// Mitsubishi GX Works2 project: may ver1   PLC: FX3G

PROGRAM MAIN
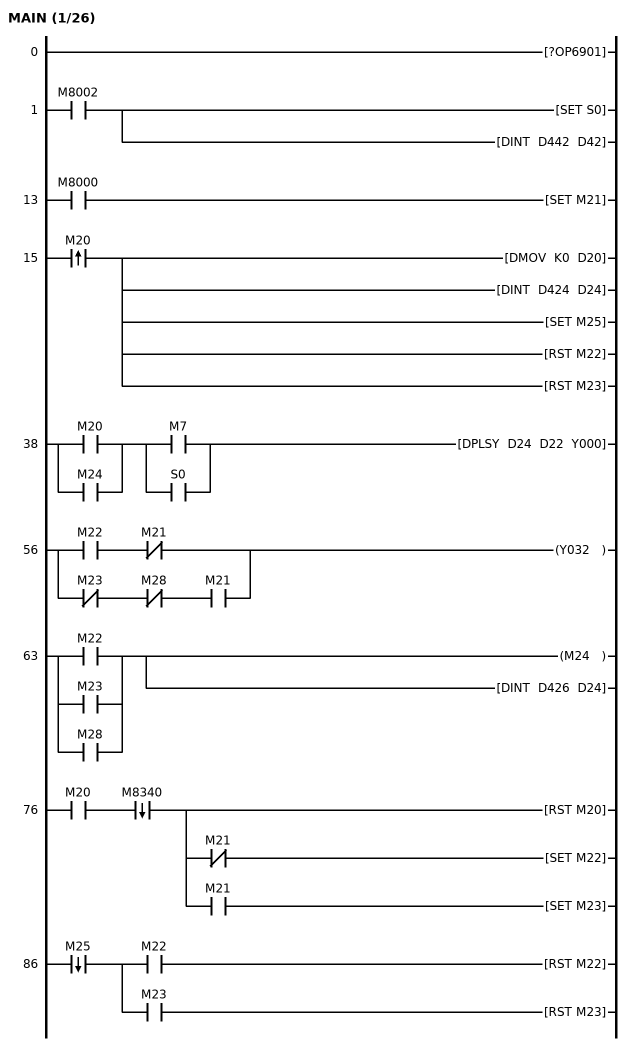
0     ?OP6901
1     LD      M8002
      SET     S0
      DINT    D442 D42
13    LD      M8000
      SET     M21
15    LDP     M20
      DMOV    K0 D20
      DINT    D424 D24
      SET     M25
      RST     M22
      RST     M23
38    LD      M20
      OR      M24
      LD      M7
      OR      S0
      ANB
      DPLSY   D24 D22 Y000
56    LD      M22
      ANI     M21
      LDI     M23
      ANI     M28
      AND     M21
      ORB
      OUT     Y032
63    LD      M22
      OR      M23
      OR      M28
      OUT     M24
      DINT    D426 D24
76    LD      M20
      ANDF    M8340
      RST     M20
      MPS
      ANI     M21
      SET     M22
      MPP
      AND     M21
      SET     M23
86    LDF     M25
      MPS
      AND     M22
      RST     M22
      MPP
      AND     M23
      RST     M23
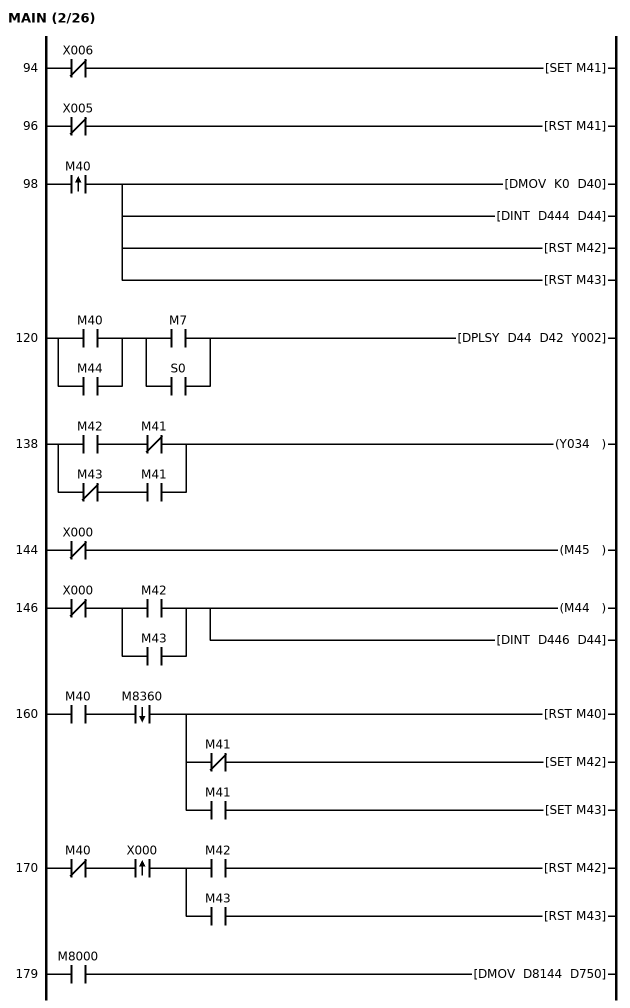
94    LDI     X006
      SET     M41
96    LDI     X005
      RST     M41
98    LDP     M40
      DMOV    K0 D40
      DINT    D444 D44
      RST     M42
      RST     M43
120   LD      M40
      OR      M44
      LD      M7
      OR      S0
      ANB
      DPLSY   D44 D42 Y002
138   LD      M42
      ANI     M41
      LDI     M43
      AND     M41
      ORB
      OUT     Y034
144   LDI     X000
      OUT     M45
146   LDI     X000
      LD      M42
      OR      M43
      ANB
      OUT     M44
      DINT    D446 D44
160   LD      M40
      ANDF    M8360
      RST     M40
      MPS
      ANI     M41
      SET     M42
      MPP
      AND     M41
      SET     M43
170   LDI     M40
      ANDP    X000
      MPS
      AND     M42
      RST     M42
      MPP
      AND     M43
      RST     M43
179   LD      M8000
      DMOV    D8144 D750
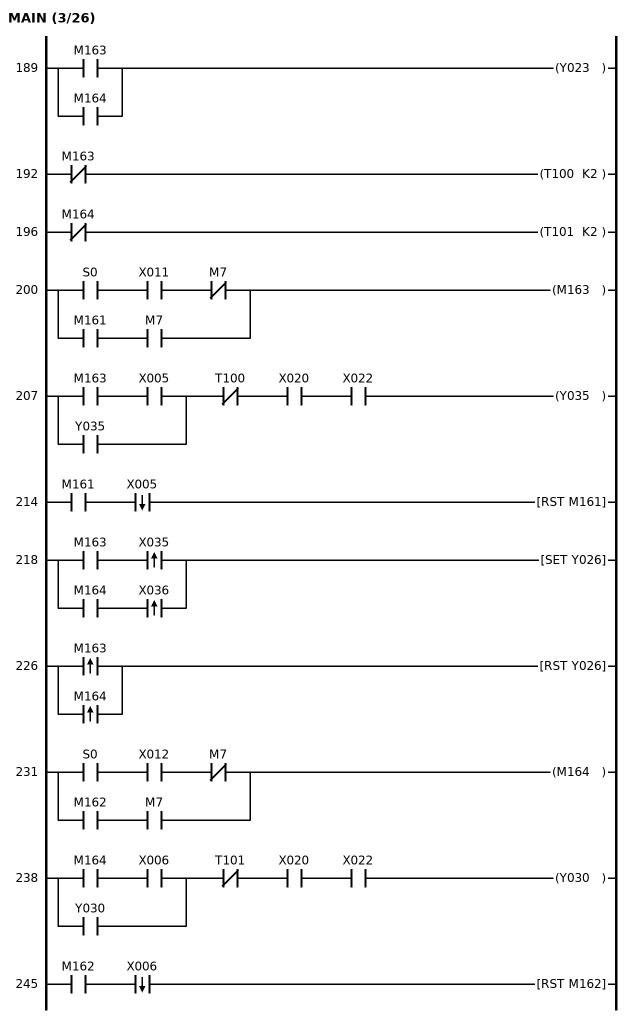
189   LD      M163
      OR      M164
      OUT     Y023
192   LDI     M163
      OUT     T100 K2
196   LDI     M164
      OUT     T101 K2
200   LD      S0
      AND     X011
      ANI     M7
      LD      M161
      AND     M7
      ORB
      OUT     M163
207   LD      M163
      AND     X005
      OR      Y035
      ANI     T100
      AND     X020
      AND     X022
      OUT     Y035
214   LD      M161
      ANDF    X005
      RST     M161
218   LD      M163
      ANDP    X035
      LD      M164
      ANDP    X036
      ORB
      SET     Y026
226   LDP     M163
      ORP     M164
      RST     Y026
231   LD      S0
      AND     X012
      ANI     M7
      LD      M162
      AND     M7
      ORB
      OUT     M164
238   LD      M164
      AND     X006
      OR      Y030
      ANI     T101
      AND     X020
      AND     X022
      OUT     Y030
245   LD      M162
      ANDF    X006
      RST     M162
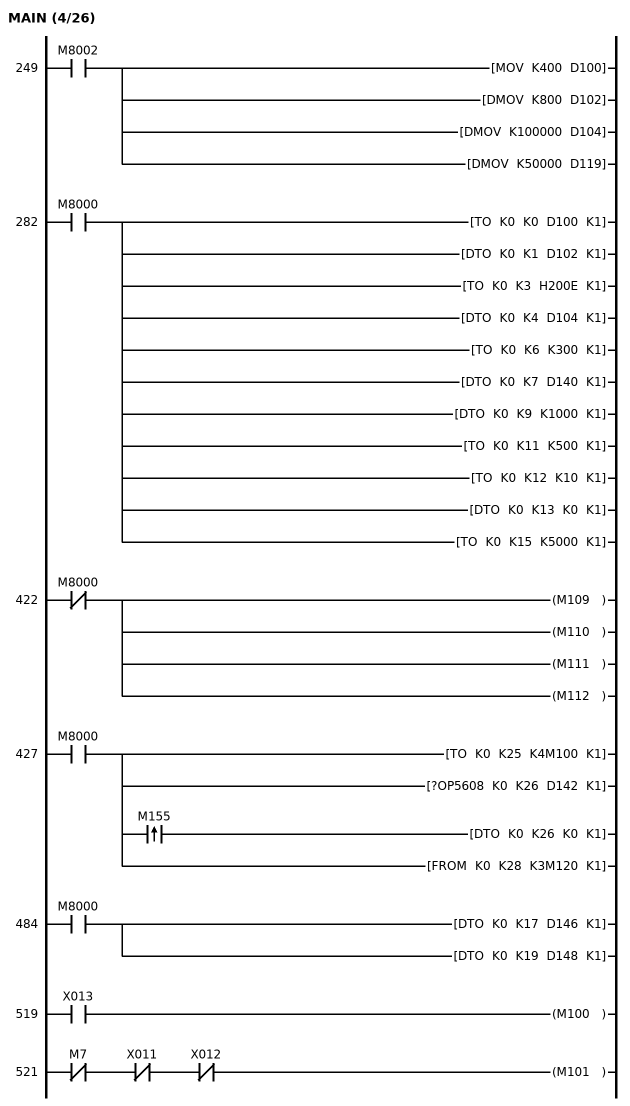
249   LD      M8002
      MOV     K400 D100
      DMOV    K800 D102
      DMOV    K100000 D104
      DMOV    K50000 D119
282   LD      M8000
      TO      K0 K0 D100 K1
      DTO     K0 K1 D102 K1
      TO      K0 K3 H200E K1
      DTO     K0 K4 D104 K1
      TO      K0 K6 K300 K1
      DTO     K0 K7 D140 K1
      DTO     K0 K9 K1000 K1
      TO      K0 K11 K500 K1
      TO      K0 K12 K10 K1
      DTO     K0 K13 K0 K1
      TO      K0 K15 K5000 K1
422   LDI     M8000
      OUT     M109
      OUT     M110
      OUT     M111
      OUT     M112
427   LD      M8000
      TO      K0 K25 K4M100 K1
      ?OP5608 K0 K26 D142 K1
      MPS
      ANDP    M155
      DTO     K0 K26 K0 K1
      MPP
      FROM    K0 K28 K3M120 K1
484   LD      M8000
      DTO     K0 K17 D146 K1
      DTO     K0 K19 D148 K1
519   LD      X013
      OUT     M100
521   LDI     M7
      ANI     X011
      ANI     X012
      OUT     M101
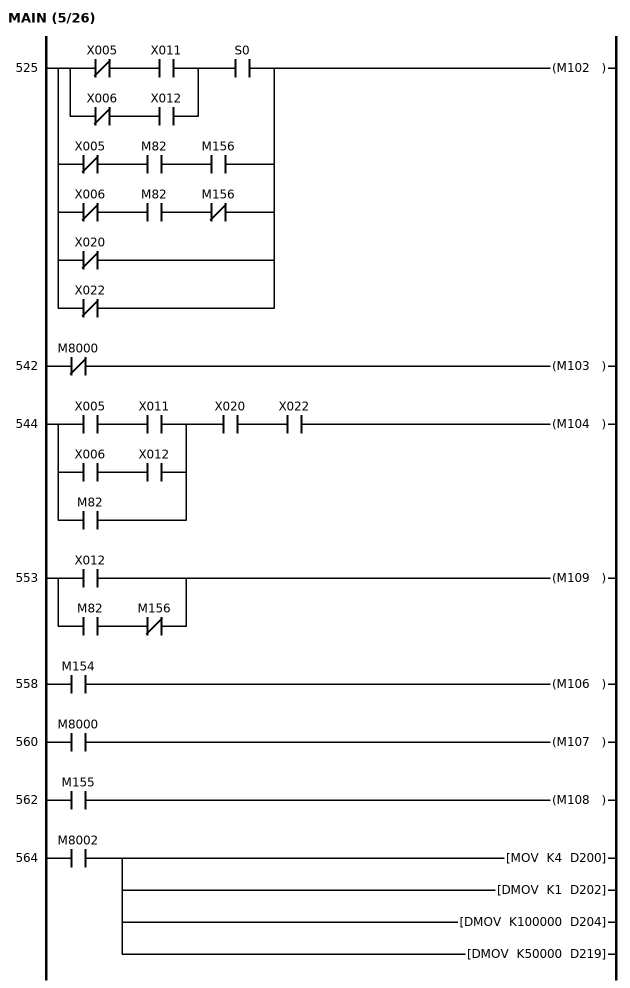
525   LDI     X005
      AND     X011
      LDI     X006
      AND     X012
      ORB
      AND     S0
      LDI     X005
      AND     M82
      AND     M156
      ORB
      LDI     X006
      AND     M82
      ANI     M156
      ORB
      ORI     X020
      ORI     X022
      OUT     M102
542   LDI     M8000
      OUT     M103
544   LD      X005
      AND     X011
      LD      X006
      AND     X012
      ORB
      OR      M82
      AND     X020
      AND     X022
      OUT     M104
553   LD      X012
      LD      M82
      ANI     M156
      ORB
      OUT     M109
558   LD      M154
      OUT     M106
560   LD      M8000
      OUT     M107
562   LD      M155
      OUT     M108
564   LD      M8002
      MOV     K4 D200
      DMOV    K1 D202
      DMOV    K100000 D204
      DMOV    K50000 D219
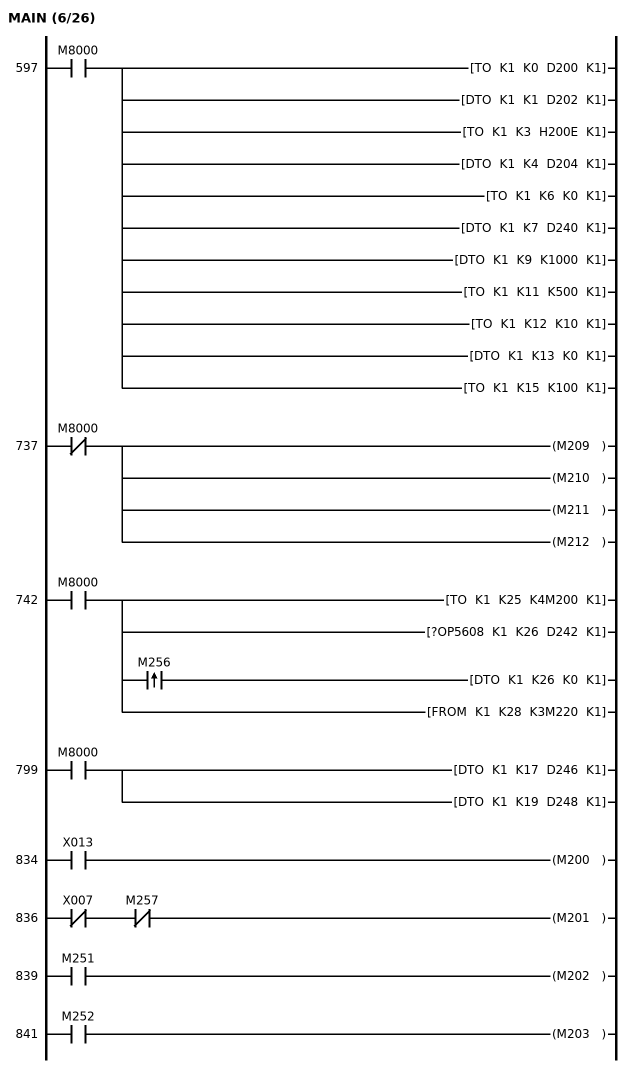
597   LD      M8000
      TO      K1 K0 D200 K1
      DTO     K1 K1 D202 K1
      TO      K1 K3 H200E K1
      DTO     K1 K4 D204 K1
      TO      K1 K6 K0 K1
      DTO     K1 K7 D240 K1
      DTO     K1 K9 K1000 K1
      TO      K1 K11 K500 K1
      TO      K1 K12 K10 K1
      DTO     K1 K13 K0 K1
      TO      K1 K15 K100 K1
737   LDI     M8000
      OUT     M209
      OUT     M210
      OUT     M211
      OUT     M212
742   LD      M8000
      TO      K1 K25 K4M200 K1
      ?OP5608 K1 K26 D242 K1
      MPS
      ANDP    M256
      DTO     K1 K26 K0 K1
      MPP
      FROM    K1 K28 K3M220 K1
799   LD      M8000
      DTO     K1 K17 D246 K1
      DTO     K1 K19 D248 K1
834   LD      X013
      OUT     M200
836   LDI     X007
      ANI     M257
      OUT     M201
839   LD      M251
      OUT     M202
841   LD      M252
      OUT     M203
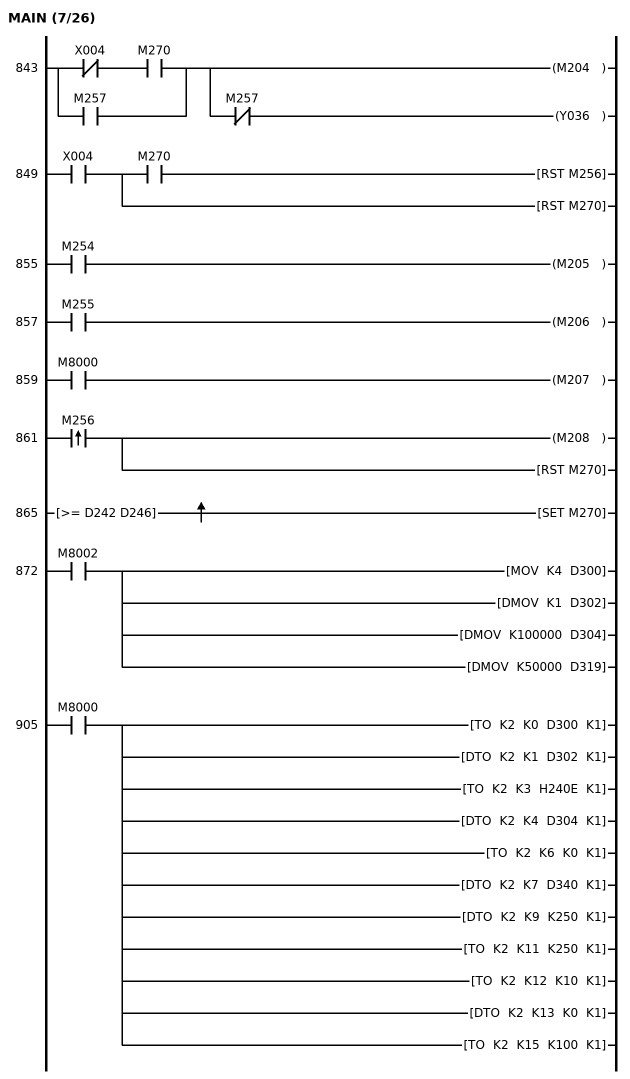
843   LDI     X004
      AND     M270
      OR      M257
      OUT     M204
      ANI     M257
      OUT     Y036
849   LD      X004
      MPS
      AND     M270
      RST     M256
      MPP
      RST     M270
855   LD      M254
      OUT     M205
857   LD      M255
      OUT     M206
859   LD      M8000
      OUT     M207
861   LDP     M256
      OUT     M208
      RST     M270
865   LD>=    D242 D246
      MEP
      SET     M270
872   LD      M8002
      MOV     K4 D300
      DMOV    K1 D302
      DMOV    K100000 D304
      DMOV    K50000 D319
905   LD      M8000
      TO      K2 K0 D300 K1
      DTO     K2 K1 D302 K1
      TO      K2 K3 H240E K1
      DTO     K2 K4 D304 K1
      TO      K2 K6 K0 K1
      DTO     K2 K7 D340 K1
      DTO     K2 K9 K250 K1
      TO      K2 K11 K250 K1
      TO      K2 K12 K10 K1
      DTO     K2 K13 K0 K1
      TO      K2 K15 K100 K1
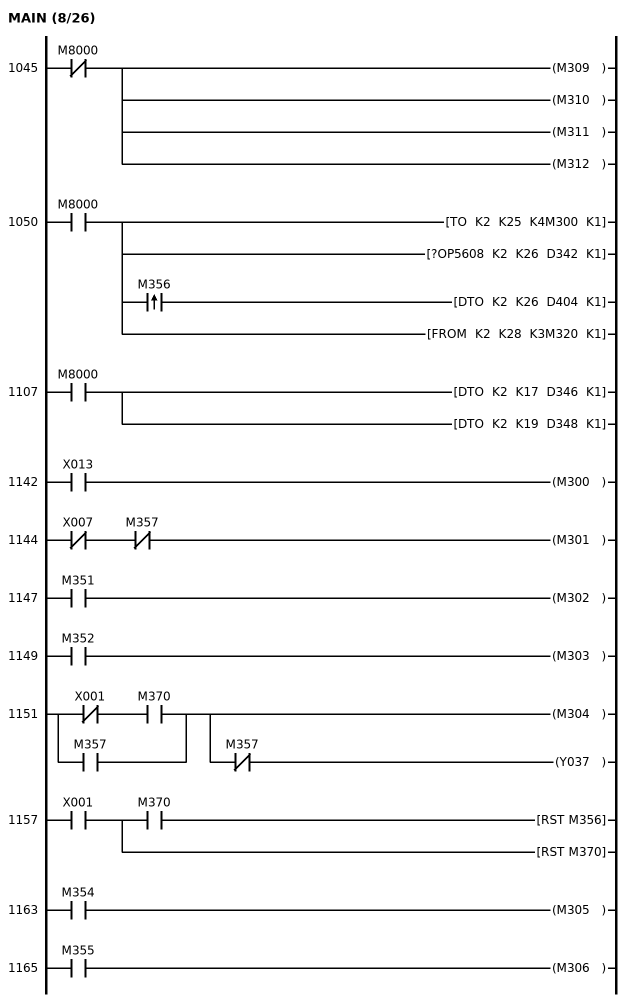
1045  LDI     M8000
      OUT     M309
      OUT     M310
      OUT     M311
      OUT     M312
1050  LD      M8000
      TO      K2 K25 K4M300 K1
      ?OP5608 K2 K26 D342 K1
      MPS
      ANDP    M356
      DTO     K2 K26 D404 K1
      MPP
      FROM    K2 K28 K3M320 K1
1107  LD      M8000
      DTO     K2 K17 D346 K1
      DTO     K2 K19 D348 K1
1142  LD      X013
      OUT     M300
1144  LDI     X007
      ANI     M357
      OUT     M301
1147  LD      M351
      OUT     M302
1149  LD      M352
      OUT     M303
1151  LDI     X001
      AND     M370
      OR      M357
      OUT     M304
      ANI     M357
      OUT     Y037
1157  LD      X001
      MPS
      AND     M370
      RST     M356
      MPP
      RST     M370
1163  LD      M354
      OUT     M305
1165  LD      M355
      OUT     M306
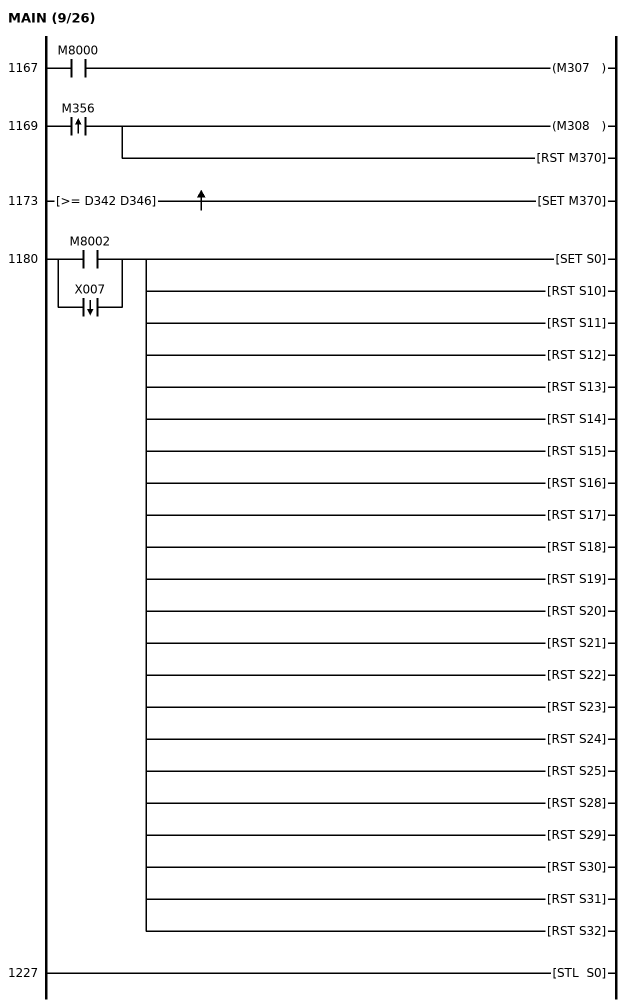
1167  LD      M8000
      OUT     M307
1169  LDP     M356
      OUT     M308
      RST     M370
1173  LD>=    D342 D346
      MEP
      SET     M370
1180  LD      M8002
      ORF     X007
      SET     S0
      RST     S10
      RST     S11
      RST     S12
      RST     S13
      RST     S14
      RST     S15
      RST     S16
      RST     S17
      RST     S18
      RST     S19
      RST     S20
      RST     S21
      RST     S22
      RST     S23
      RST     S24
      RST     S25
      RST     S28
      RST     S29
      RST     S30
      RST     S31
      RST     S32
1227  STL     S0
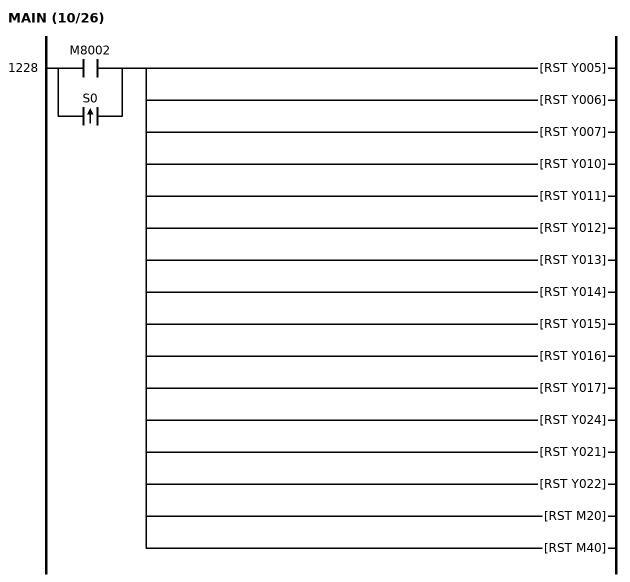
1228  LD      M8002
      ORP     S0
      RST     Y005
      RST     Y006
      RST     Y007
      RST     Y010
      RST     Y011
      RST     Y012
      RST     Y013
      RST     Y014
      RST     Y015
      RST     Y016
      RST     Y017
      RST     Y024
      RST     Y021
      RST     Y022
      RST     M20
      RST     M40
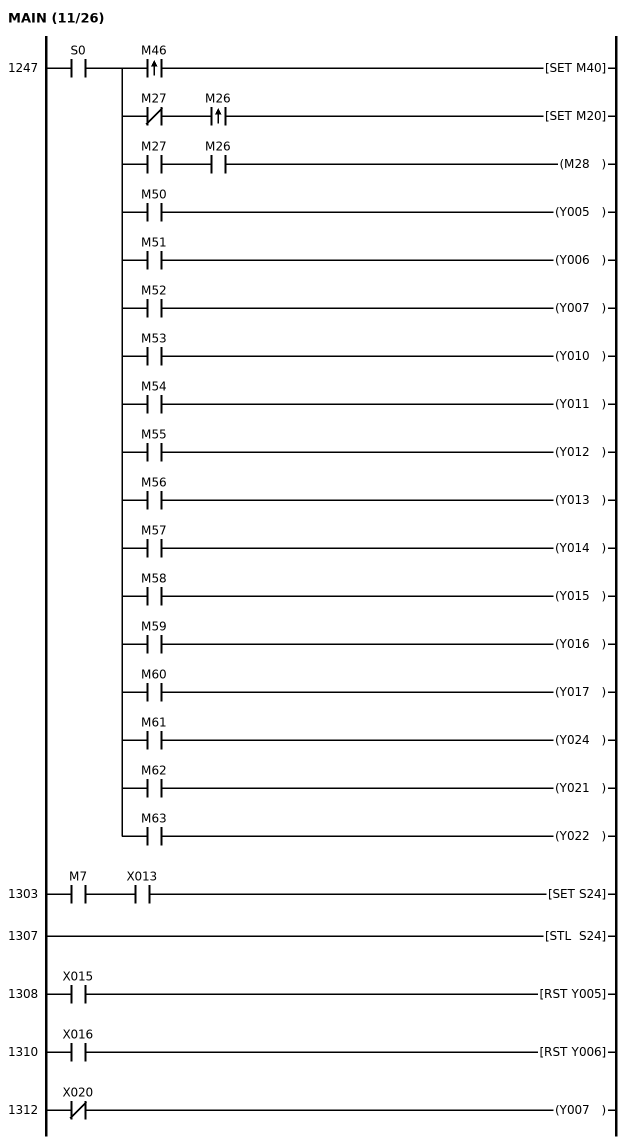
1247  LD      S0
      MPS
      ANDP    M46
      SET     M40
      MRD
      ANI     M27
      ANDP    M26
      SET     M20
      MRD
      AND     M27
      AND     M26
      OUT     M28
      MRD
      AND     M50
      OUT     Y005
      MRD
      AND     M51
      OUT     Y006
      MRD
      AND     M52
      OUT     Y007
      MRD
      AND     M53
      OUT     Y010
      MRD
      AND     M54
      OUT     Y011
      MRD
      AND     M55
      OUT     Y012
      MRD
      AND     M56
      OUT     Y013
      MRD
      AND     M57
      OUT     Y014
      MRD
      AND     M58
      OUT     Y015
      MRD
      AND     M59
      OUT     Y016
      MRD
      AND     M60
      OUT     Y017
      MRD
      AND     M61
      OUT     Y024
      MRD
      AND     M62
      OUT     Y021
      MPP
      AND     M63
      OUT     Y022
1303  LD      M7
      AND     X013
      SET     S24
1307  STL     S24
1308  LD      X015
      RST     Y005
1310  LD      X016
      RST     Y006
1312  LDI     X020
      OUT     Y007
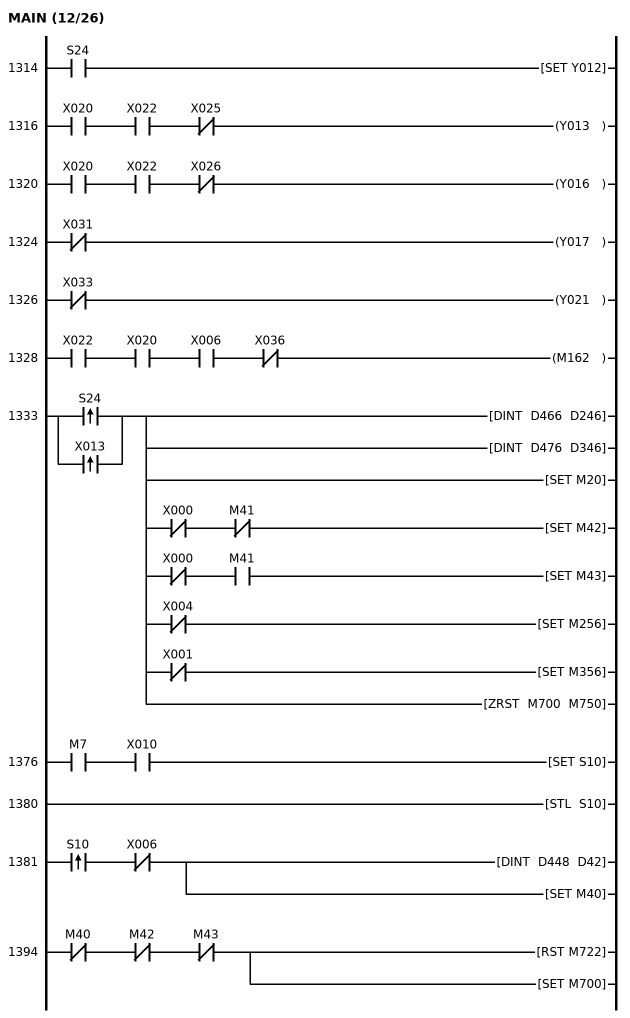
1314  LD      S24
      SET     Y012
1316  LD      X020
      AND     X022
      ANI     X025
      OUT     Y013
1320  LD      X020
      AND     X022
      ANI     X026
      OUT     Y016
1324  LDI     X031
      OUT     Y017
1326  LDI     X033
      OUT     Y021
1328  LD      X022
      AND     X020
      AND     X006
      ANI     X036
      OUT     M162
1333  LDP     S24
      ORP     X013
      DINT    D466 D246
      DINT    D476 D346
      SET     M20
      MPS
      ANI     X000
      ANI     M41
      SET     M42
      MRD
      ANI     X000
      AND     M41
      SET     M43
      MRD
      ANI     X004
      SET     M256
      MRD
      ANI     X001
      SET     M356
      MPP
      ZRST    M700 M750
1376  LD      M7
      AND     X010
      SET     S10
1380  STL     S10
1381  LDP     S10
      ANI     X006
      DINT    D448 D42
      SET     M40
1394  LDI     M40
      ANI     M42
      ANI     M43
      RST     M722
      SET     M700
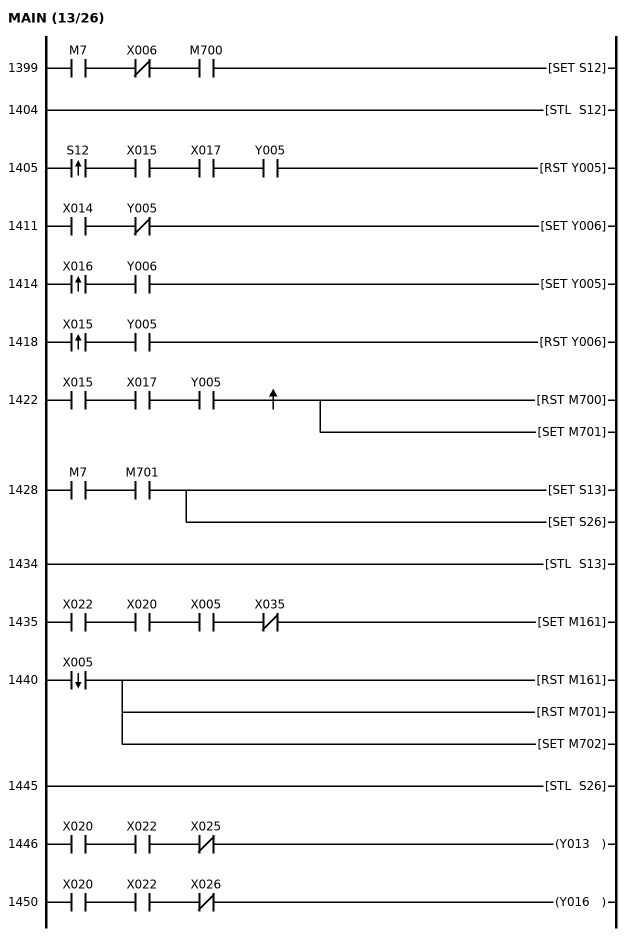
1399  LD      M7
      ANI     X006
      AND     M700
      SET     S12
1404  STL     S12
1405  LDP     S12
      AND     X015
      AND     X017
      AND     Y005
      RST     Y005
1411  LD      X014
      ANI     Y005
      SET     Y006
1414  LDP     X016
      AND     Y006
      SET     Y005
1418  LDP     X015
      AND     Y005
      RST     Y006
1422  LD      X015
      AND     X017
      AND     Y005
      MEP
      RST     M700
      SET     M701
1428  LD      M7
      AND     M701
      SET     S13
      SET     S26
1434  STL     S13
1435  LD      X022
      AND     X020
      AND     X005
      ANI     X035
      SET     M161
1440  LDF     X005
      RST     M161
      RST     M701
      SET     M702
1445  STL     S26
1446  LD      X020
      AND     X022
      ANI     X025
      OUT     Y013
1450  LD      X020
      AND     X022
      ANI     X026
      OUT     Y016
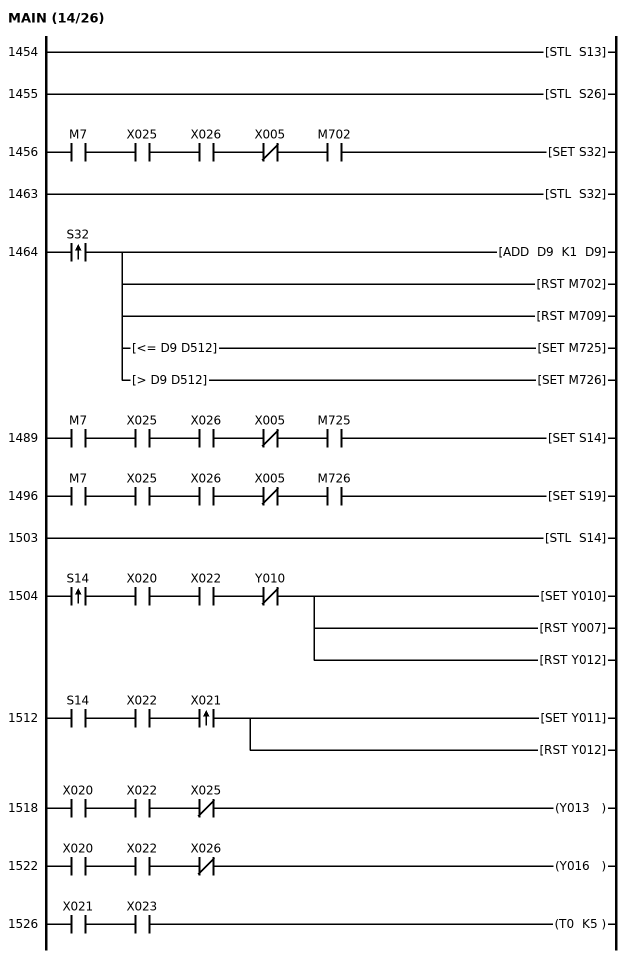
1454  STL     S13
1455  STL     S26
1456  LD      M7
      AND     X025
      AND     X026
      ANI     X005
      AND     M702
      SET     S32
1463  STL     S32
1464  LDP     S32
      ADD     D9 K1 D9
      RST     M702
      RST     M709
      MPS
      AND<=   D9 D512
      SET     M725
      MPP
      AND>    D9 D512
      SET     M726
1489  LD      M7
      AND     X025
      AND     X026
      ANI     X005
      AND     M725
      SET     S14
1496  LD      M7
      AND     X025
      AND     X026
      ANI     X005
      AND     M726
      SET     S19
1503  STL     S14
1504  LDP     S14
      AND     X020
      AND     X022
      ANI     Y010
      SET     Y010
      RST     Y007
      RST     Y012
1512  LD      S14
      AND     X022
      ANDP    X021
      SET     Y011
      RST     Y012
1518  LD      X020
      AND     X022
      ANI     X025
      OUT     Y013
1522  LD      X020
      AND     X022
      ANI     X026
      OUT     Y016
1526  LD      X021
      AND     X023
      OUT     T0 K5
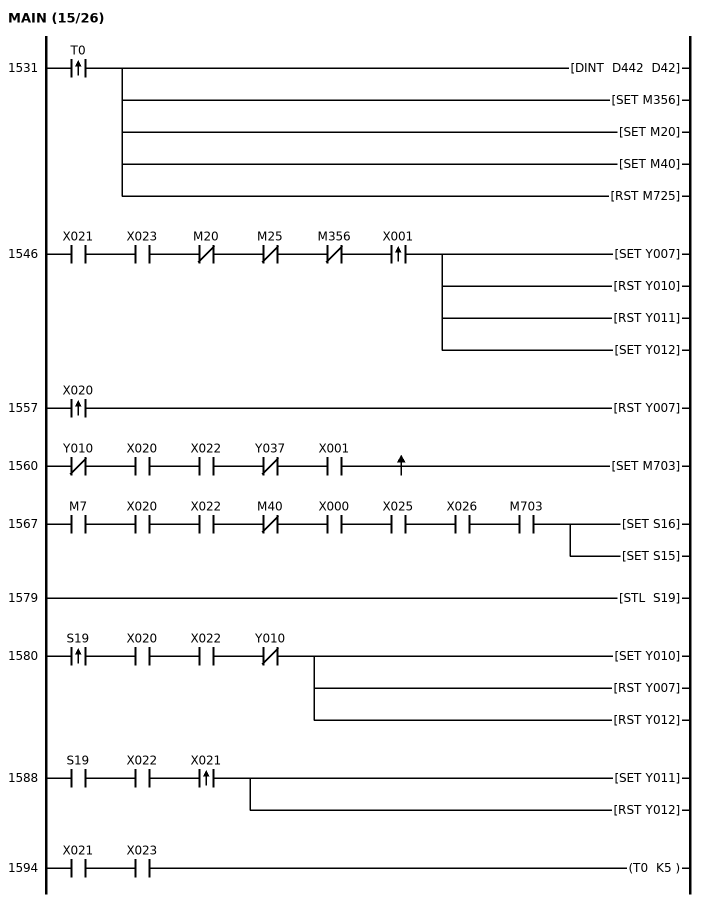
1531  LDP     T0
      DINT    D442 D42
      SET     M356
      SET     M20
      SET     M40
      RST     M725
1546  LD      X021
      AND     X023
      ANI     M20
      ANI     M25
      ANI     M356
      ANDP    X001
      SET     Y007
      RST     Y010
      RST     Y011
      SET     Y012
1557  LDP     X020
      RST     Y007
1560  LDI     Y010
      AND     X020
      AND     X022
      ANI     Y037
      AND     X001
      MEP
      SET     M703
1567  LD      M7
      AND     X020
      AND     X022
      ANI     M40
      AND     X000
      AND     X025
      AND     X026
      AND     M703
      SET     S16
      SET     S15
1579  STL     S19
1580  LDP     S19
      AND     X020
      AND     X022
      ANI     Y010
      SET     Y010
      RST     Y007
      RST     Y012
1588  LD      S19
      AND     X022
      ANDP    X021
      SET     Y011
      RST     Y012
1594  LD      X021
      AND     X023
      OUT     T0 K5
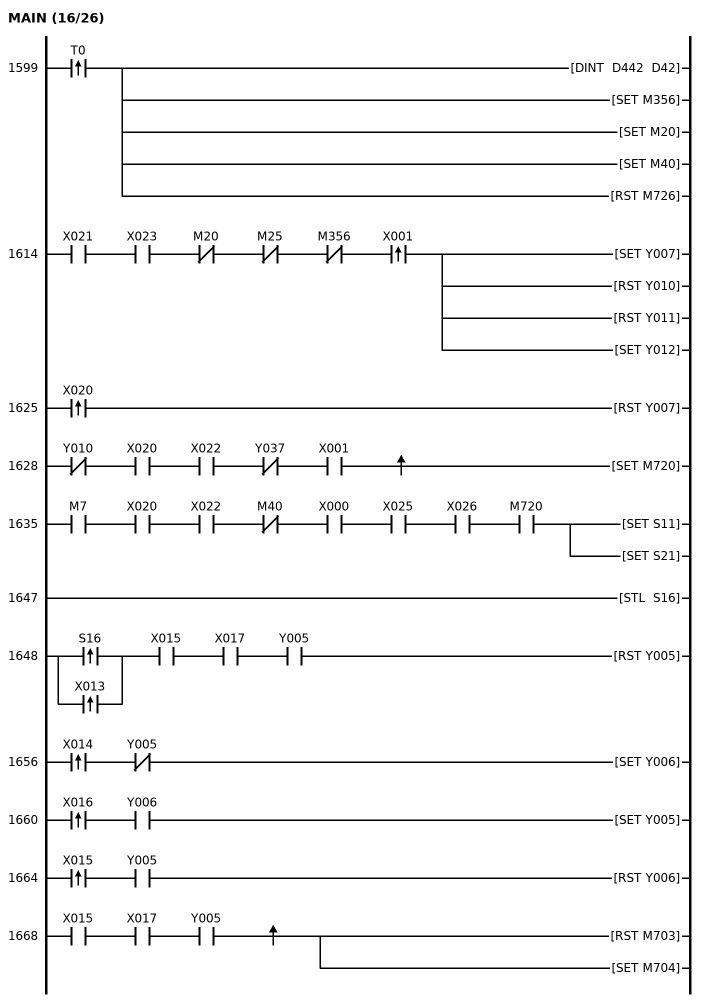
1599  LDP     T0
      DINT    D442 D42
      SET     M356
      SET     M20
      SET     M40
      RST     M726
1614  LD      X021
      AND     X023
      ANI     M20
      ANI     M25
      ANI     M356
      ANDP    X001
      SET     Y007
      RST     Y010
      RST     Y011
      SET     Y012
1625  LDP     X020
      RST     Y007
1628  LDI     Y010
      AND     X020
      AND     X022
      ANI     Y037
      AND     X001
      MEP
      SET     M720
1635  LD      M7
      AND     X020
      AND     X022
      ANI     M40
      AND     X000
      AND     X025
      AND     X026
      AND     M720
      SET     S11
      SET     S21
1647  STL     S16
1648  LDP     S16
      ORP     X013
      AND     X015
      AND     X017
      AND     Y005
      RST     Y005
1656  LDP     X014
      ANI     Y005
      SET     Y006
1660  LDP     X016
      AND     Y006
      SET     Y005
1664  LDP     X015
      AND     Y005
      RST     Y006
1668  LD      X015
      AND     X017
      AND     Y005
      MEP
      RST     M703
      SET     M704
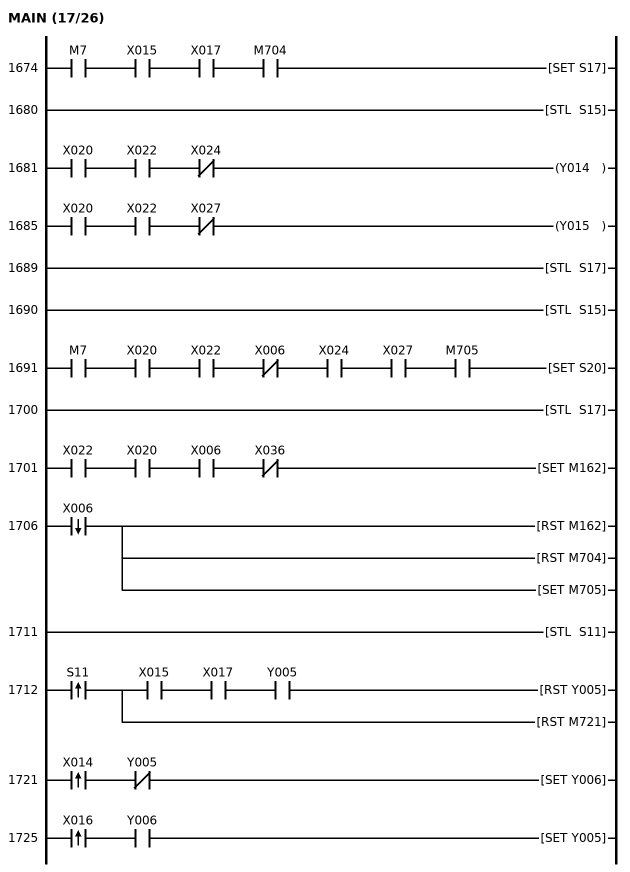
1674  LD      M7
      AND     X015
      AND     X017
      AND     M704
      SET     S17
1680  STL     S15
1681  LD      X020
      AND     X022
      ANI     X024
      OUT     Y014
1685  LD      X020
      AND     X022
      ANI     X027
      OUT     Y015
1689  STL     S17
1690  STL     S15
1691  LD      M7
      AND     X020
      AND     X022
      ANI     X006
      AND     X024
      AND     X027
      AND     M705
      SET     S20
1700  STL     S17
1701  LD      X022
      AND     X020
      AND     X006
      ANI     X036
      SET     M162
1706  LDF     X006
      RST     M162
      RST     M704
      SET     M705
1711  STL     S11
1712  LDP     S11
      MPS
      AND     X015
      AND     X017
      AND     Y005
      RST     Y005
      MPP
      RST     M721
1721  LDP     X014
      ANI     Y005
      SET     Y006
1725  LDP     X016
      AND     Y006
      SET     Y005
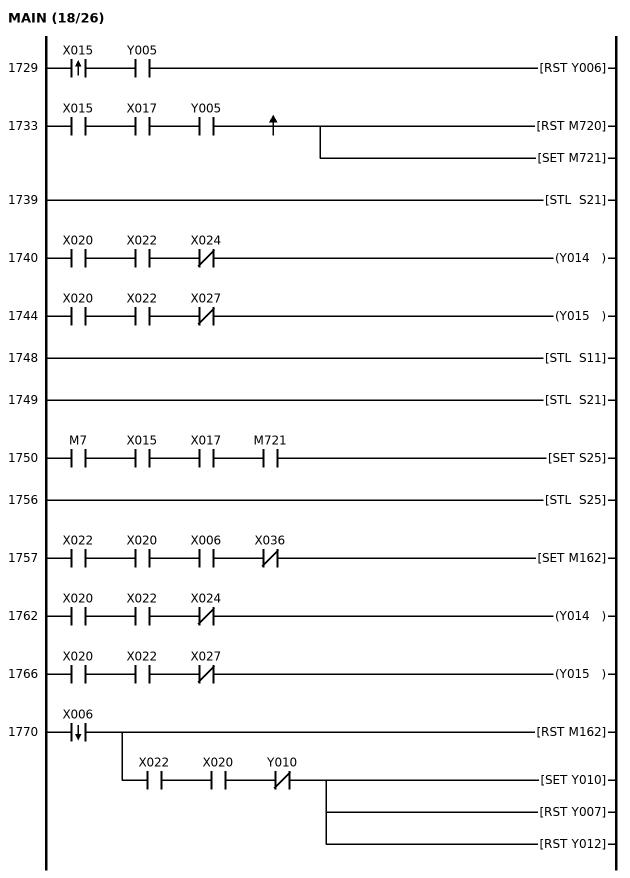
1729  LDP     X015
      AND     Y005
      RST     Y006
1733  LD      X015
      AND     X017
      AND     Y005
      MEP
      RST     M720
      SET     M721
1739  STL     S21
1740  LD      X020
      AND     X022
      ANI     X024
      OUT     Y014
1744  LD      X020
      AND     X022
      ANI     X027
      OUT     Y015
1748  STL     S11
1749  STL     S21
1750  LD      M7
      AND     X015
      AND     X017
      AND     M721
      SET     S25
1756  STL     S25
1757  LD      X022
      AND     X020
      AND     X006
      ANI     X036
      SET     M162
1762  LD      X020
      AND     X022
      ANI     X024
      OUT     Y014
1766  LD      X020
      AND     X022
      ANI     X027
      OUT     Y015
1770  LDF     X006
      RST     M162
      AND     X022
      AND     X020
      ANI     Y010
      SET     Y010
      RST     Y007
      RST     Y012
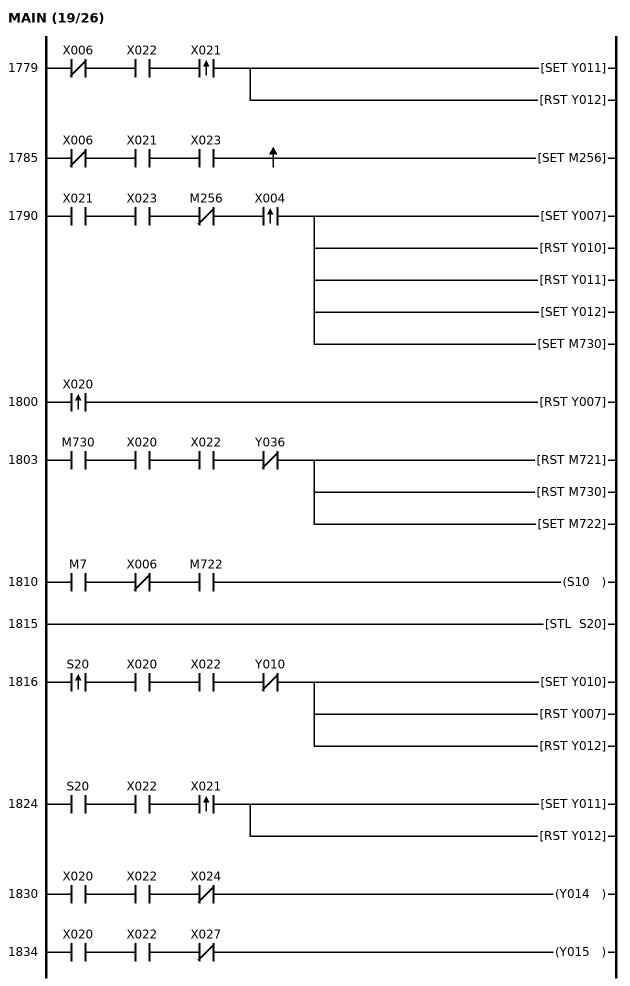
1779  LDI     X006
      AND     X022
      ANDP    X021
      SET     Y011
      RST     Y012
1785  LDI     X006
      AND     X021
      AND     X023
      MEP
      SET     M256
1790  LD      X021
      AND     X023
      ANI     M256
      ANDP    X004
      SET     Y007
      RST     Y010
      RST     Y011
      SET     Y012
      SET     M730
1800  LDP     X020
      RST     Y007
1803  LD      M730
      AND     X020
      AND     X022
      ANI     Y036
      RST     M721
      RST     M730
      SET     M722
1810  LD      M7
      ANI     X006
      AND     M722
      OUT     S10
1815  STL     S20
1816  LDP     S20
      AND     X020
      AND     X022
      ANI     Y010
      SET     Y010
      RST     Y007
      RST     Y012
1824  LD      S20
      AND     X022
      ANDP    X021
      SET     Y011
      RST     Y012
1830  LD      X020
      AND     X022
      ANI     X024
      OUT     Y014
1834  LD      X020
      AND     X022
      ANI     X027
      OUT     Y015
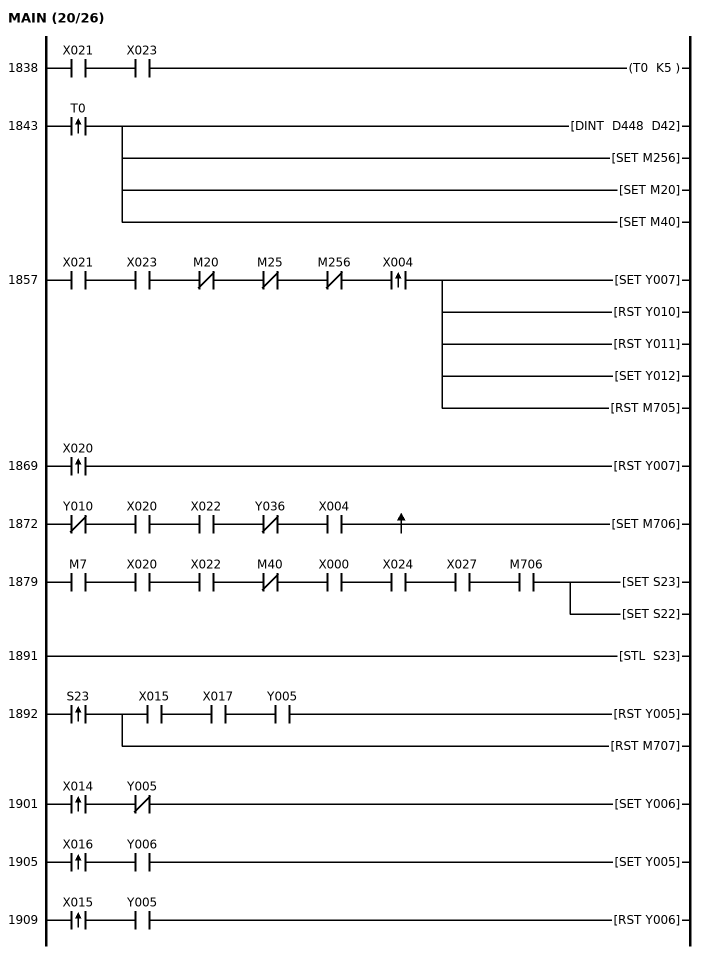
1838  LD      X021
      AND     X023
      OUT     T0 K5
1843  LDP     T0
      DINT    D448 D42
      SET     M256
      SET     M20
      SET     M40
1857  LD      X021
      AND     X023
      ANI     M20
      ANI     M25
      ANI     M256
      ANDP    X004
      SET     Y007
      RST     Y010
      RST     Y011
      SET     Y012
      RST     M705
1869  LDP     X020
      RST     Y007
1872  LDI     Y010
      AND     X020
      AND     X022
      ANI     Y036
      AND     X004
      MEP
      SET     M706
1879  LD      M7
      AND     X020
      AND     X022
      ANI     M40
      AND     X000
      AND     X024
      AND     X027
      AND     M706
      SET     S23
      SET     S22
1891  STL     S23
1892  LDP     S23
      MPS
      AND     X015
      AND     X017
      AND     Y005
      RST     Y005
      MPP
      RST     M707
1901  LDP     X014
      ANI     Y005
      SET     Y006
1905  LDP     X016
      AND     Y006
      SET     Y005
1909  LDP     X015
      AND     Y005
      RST     Y006
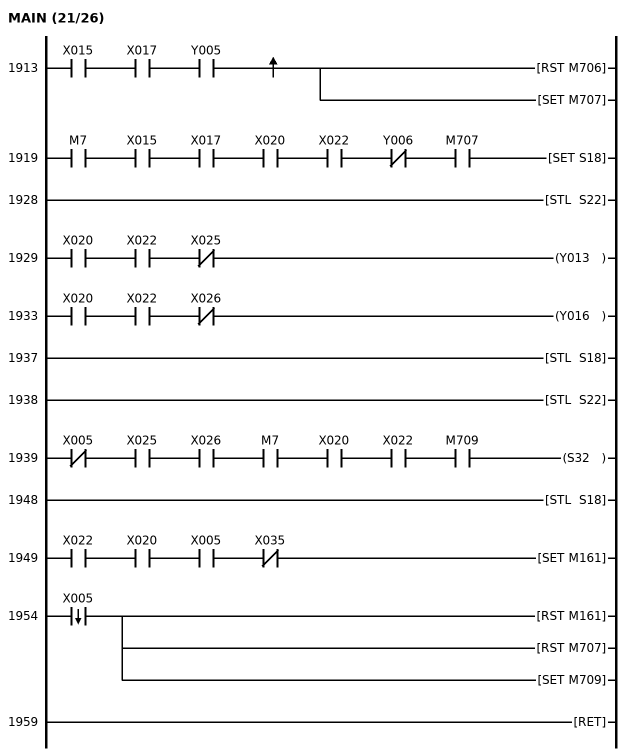
1913  LD      X015
      AND     X017
      AND     Y005
      MEP
      RST     M706
      SET     M707
1919  LD      M7
      AND     X015
      AND     X017
      AND     X020
      AND     X022
      ANI     Y006
      AND     M707
      SET     S18
1928  STL     S22
1929  LD      X020
      AND     X022
      ANI     X025
      OUT     Y013
1933  LD      X020
      AND     X022
      ANI     X026
      OUT     Y016
1937  STL     S18
1938  STL     S22
1939  LDI     X005
      AND     X025
      AND     X026
      AND     M7
      AND     X020
      AND     X022
      AND     M709
      OUT     S32
1948  STL     S18
1949  LD      X022
      AND     X020
      AND     X005
      ANI     X035
      SET     M161
1954  LDF     X005
      RST     M161
      RST     M707
      SET     M709
1959  RET
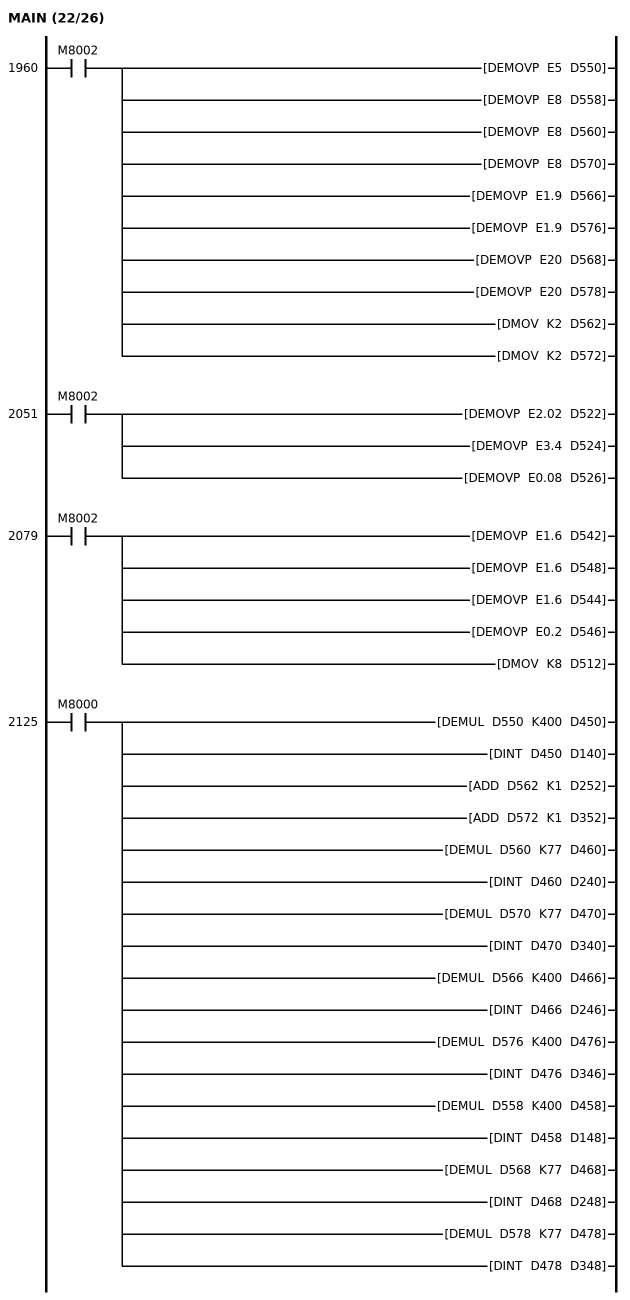
1960  LD      M8002
      DEMOVP  E5 D550
      DEMOVP  E8 D558
      DEMOVP  E8 D560
      DEMOVP  E8 D570
      DEMOVP  E1.9 D566
      DEMOVP  E1.9 D576
      DEMOVP  E20 D568
      DEMOVP  E20 D578
      DMOV    K2 D562
      DMOV    K2 D572
2051  LD      M8002
      DEMOVP  E2.02 D522
      DEMOVP  E3.4 D524
      DEMOVP  E0.08 D526
2079  LD      M8002
      DEMOVP  E1.6 D542
      DEMOVP  E1.6 D548
      DEMOVP  E1.6 D544
      DEMOVP  E0.2 D546
      DMOV    K8 D512
2125  LD      M8000
      DEMUL   D550 K400 D450
      DINT    D450 D140
      ADD     D562 K1 D252
      ADD     D572 K1 D352
      DEMUL   D560 K77 D460
      DINT    D460 D240
      DEMUL   D570 K77 D470
      DINT    D470 D340
      DEMUL   D566 K400 D466
      DINT    D466 D246
      DEMUL   D576 K400 D476
      DINT    D476 D346
      DEMUL   D558 K400 D458
      DINT    D458 D148
      DEMUL   D568 K77 D468
      DINT    D468 D248
      DEMUL   D578 K77 D478
      DINT    D478 D348
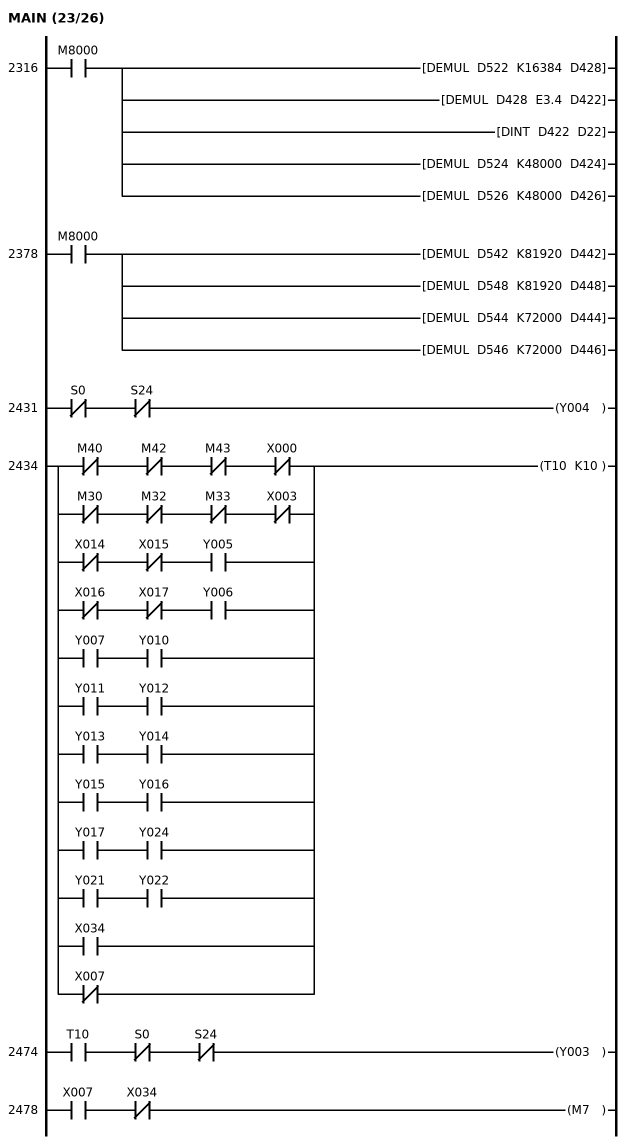
2316  LD      M8000
      DEMUL   D522 K16384 D428
      DEMUL   D428 E3.4 D422
      DINT    D422 D22
      DEMUL   D524 K48000 D424
      DEMUL   D526 K48000 D426
2378  LD      M8000
      DEMUL   D542 K81920 D442
      DEMUL   D548 K81920 D448
      DEMUL   D544 K72000 D444
      DEMUL   D546 K72000 D446
2431  LDI     S0
      ANI     S24
      OUT     Y004
2434  LDI     M40
      ANI     M42
      ANI     M43
      ANI     X000
      LDI     M30
      ANI     M32
      ANI     M33
      ANI     X003
      ORB
      LDI     X014
      ANI     X015
      AND     Y005
      ORB
      LDI     X016
      ANI     X017
      AND     Y006
      ORB
      LD      Y007
      AND     Y010
      ORB
      LD      Y011
      AND     Y012
      ORB
      LD      Y013
      AND     Y014
      ORB
      LD      Y015
      AND     Y016
      ORB
      LD      Y017
      AND     Y024
      ORB
      LD      Y021
      AND     Y022
      ORB
      OR      X034
      ORI     X007
      OUT     T10 K10
2474  LD      T10
      ANI     S0
      ANI     S24
      OUT     Y003
2478  LD      X007
      ANI     X034
      OUT     M7
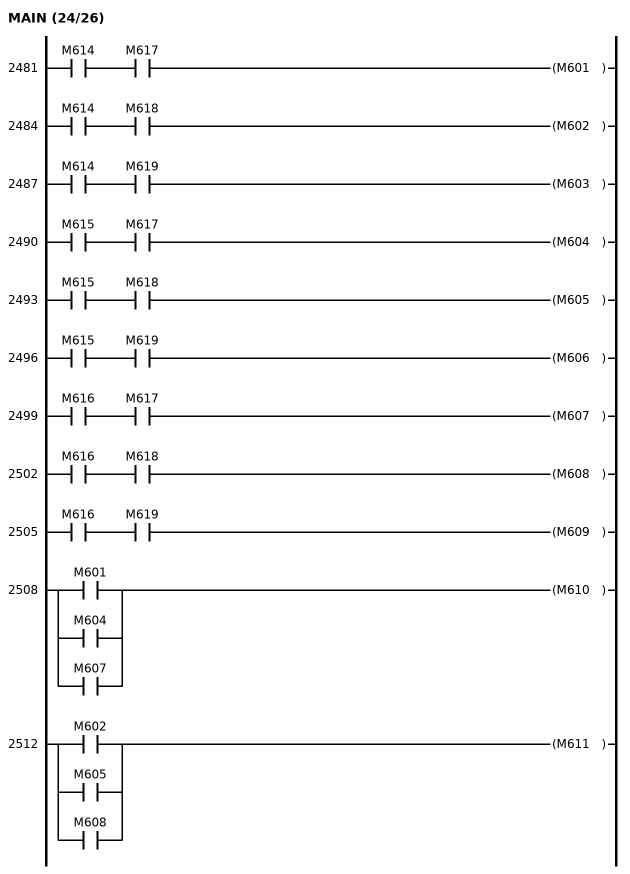
2481  LD      M614
      AND     M617
      OUT     M601
2484  LD      M614
      AND     M618
      OUT     M602
2487  LD      M614
      AND     M619
      OUT     M603
2490  LD      M615
      AND     M617
      OUT     M604
2493  LD      M615
      AND     M618
      OUT     M605
2496  LD      M615
      AND     M619
      OUT     M606
2499  LD      M616
      AND     M617
      OUT     M607
2502  LD      M616
      AND     M618
      OUT     M608
2505  LD      M616
      AND     M619
      OUT     M609
2508  LD      M601
      OR      M604
      OR      M607
      OUT     M610
2512  LD      M602
      OR      M605
      OR      M608
      OUT     M611
